{attribute 'enable_dynamic_creation'}
FUNCTION_BLOCK FutureMCGearOut EXTENDS FB_AbstructFuture
VAR_INPUT
END_VAR
VAR_OUTPUT
END_VAR
VAR
	_fb_gear_out	: MC_GearOut;
	_mc_reset	: MC_Reset;
	_axis_sub: REFERENCE TO AXIS_REF;
	_ratio_numerator	: MC_LREAL := 1;
	_ratio_denominator	: UINT := 1;
	_option : ST_GearOutOptions;
	_error_id :HRESULT;
	_exec_state : UDINT;
END_VAR

METHOD error_reset : BOOL // Must be overrided if future has any errors.
IF _error_id <> 0 THEN
	CASE _exec_state OF
		0:
			_mc_reset(Axis := _axis_sub, Execute := FALSE);
			_mc_reset(Axis:= _axis_sub, Execute := TRUE );
			_exec_state := 1;
		1:
			IF _mc_reset.Busy THEN
				_mc_reset(Axis:= _axis_sub,Execute := FALSE);
			END_IF
	END_CASE
	
	_error_id := _mc_reset.ErrorID;
	error_reset := _mc_reset.Done;
ELSE
	error_reset := TRUE;
END_IF
END_METHOD

METHOD execute : BOOL // Return TRUE if finish.
execute := FALSE;
CASE _exec_state OF
	0:
		_fb_gear_out(Slave := _axis_sub,Execute := FALSE);
		_fb_gear_out(
			Execute := TRUE,
			Slave := _axis_sub,
			Options := _option
		);
		_exec_state := 1;
	1:
		IF _fb_gear_out.Busy THEN
			_fb_gear_out(Slave := _axis_sub,Execute := FALSE);
		END_IF
		IF NOT _fb_gear_out.Execute AND NOT _fb_gear_out.Busy THEN
			_exec_state := 2;
		END_IF
	2:
		IF _fb_gear_out.Done OR _fb_gear_out.Error THEN
			_exec_state := 3;
		END_IF
	3:
		execute := TRUE;
		
END_CASE

_error_id := _fb_gear_out.ErrorID;
END_METHOD

METHOD init : BOOL // Return TRUE if finish.

VAR
	axis: INT;
END_VAR
_exec_state := 0;
_error_id := _fb_gear_out.ErrorID;
init := TRUE;
END_METHOD

PROPERTY nErrorID : HRESULT
GET
nErrorID := _error_id;
END_GET
SET
END_SET
END_PROPERTY

METHOD set_options : BOOL
VAR_INPUT
	option : ST_GearOutOptions;
END_VAR
_option := option;
END_METHOD

METHOD set_parameters : BOOL
VAR_INPUT
	axis_sub : REFERENCE TO AXIS_REF;
END_VAR
_axis_sub REF= axis_sub;
END_METHOD

END_FUNCTION_BLOCK

(* stored: Version 1.1.0.1, ProductVersion 3.1.4026.13
   POU FutureMCGearOut: Id {b10cbfcd-3f21-4d41-b1d5-2cbad711776c}, SpecialFunc None
   Method error_reset: Id {52e60225-068f-4e49-a10a-be6c8142996b}
   Method execute: Id {10b8fb9d-57b5-428e-b814-1bfc496da251}
   Method init: Id {7dc29fac-86ad-4c32-8e88-fd323e0c0da2}
   Property nErrorID: Id {c7ba103c-81cf-4b3f-83df-e6c1e7846eb9}
   Get Get: Id {71af881f-7335-458d-a52b-3bf08345a0cc}
   Set Set: Id {00e1a2d2-86de-4ef0-806d-26a546c23421}
   Method set_options: Id {22525b5f-688d-4193-806d-a7ceed51892e}
   Method set_parameters: Id {9e93cc8f-23ba-4f40-9f9d-19dd7cdae208} *)
